% RSLogix 500 project TestPLC.RSS, saved by version 9.00.00.04 %
PROJECT "UNTITLED"    % processor: MicroLogix 1400 %

PROGRAM FILES
  LAD 2   17 rungs

DATA FILES
  O0 OUTPUT  6 elements
  I1 INPUT  8 elements
  S2 STATUS  66 elements
  B3 BINARY  3 elements
  T4 TIMER  3 elements
  C5 COUNTER  1 elements
  R6 CONTROL  1 elements
  N7 INTEGER  10 elements
  F8 FLOAT  3 elements
  N9 BATCH  11 elements  % store btch numbers %
  RI10   1 elements
  MG11 CREATESOCK  2 elements
  MG13   1 elements
  RI14   1 elements
  RI40   15 elements

LADDER 2
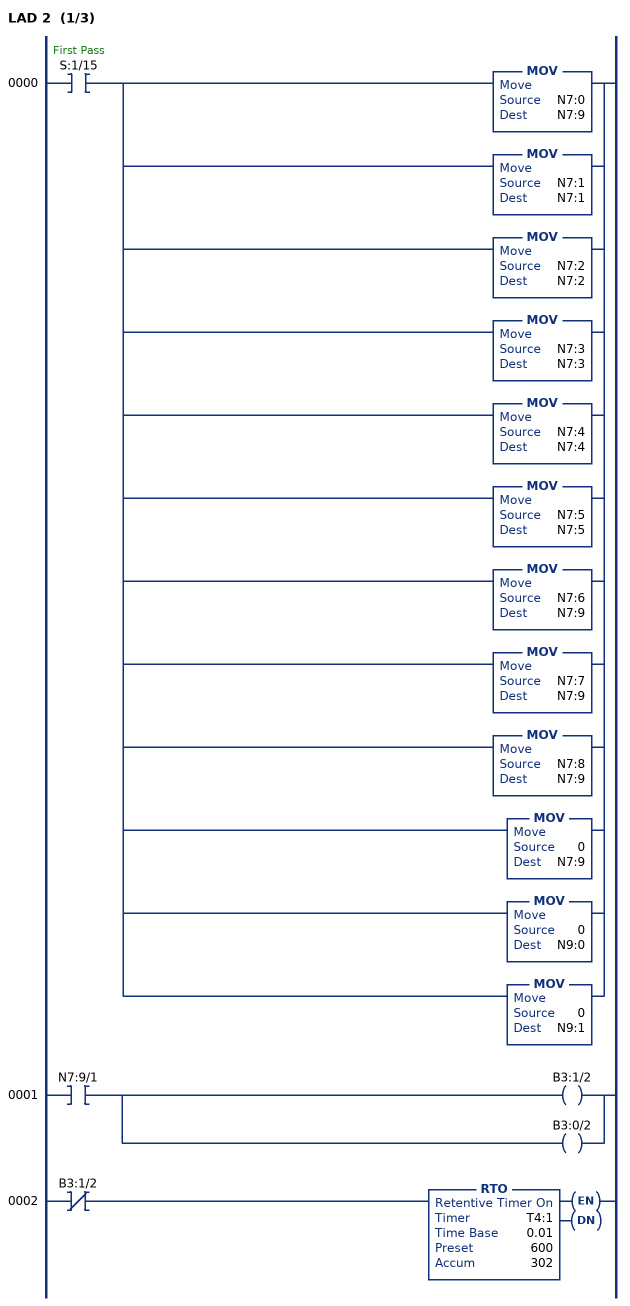
% Rung: 0 %
SOR XIC S:1/15 BST MOV N7:0 N7:9 NXB MOV N7:1 N7:1 NXB MOV N7:2 N7:2 NXB MOV N7:3 N7:3 NXB MOV N7:4 N7:4 NXB MOV N7:5 N7:5 NXB MOV N7:6 N7:9 NXB MOV N7:7 N7:9 NXB MOV N7:8 N7:9 NXB MOV 0 N7:9 NXB MOV 0 N9:0 NXB MOV 0 N9:1 BND EOR
%   S:1/15  "First Pass" %
%   N7:0  "Clr Control Block" %
% Rung: 1 %
SOR XIC N7:9/1 BST OTE B3:1/2 NXB OTE B3:0/2 BND EOR
% Rung: 2 %
SOR XIO B3:1/2 RTO T4:1 0.01 600 302 EOR

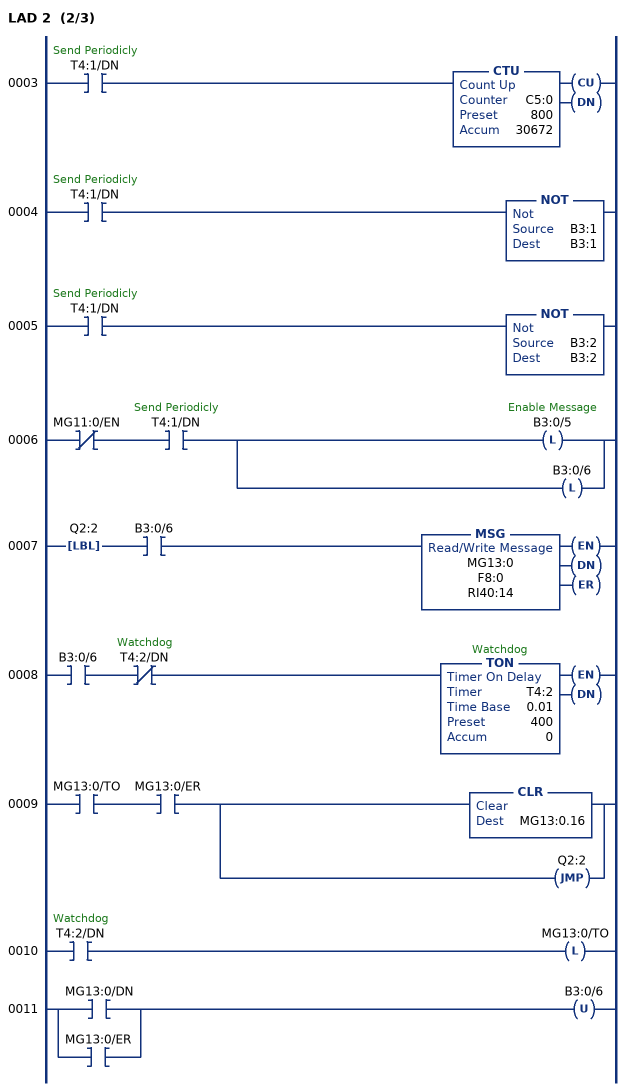
% Rung: 3 %
SOR XIC T4:1/DN CTU C5:0 800 30672 EOR
%   T4:1/DN  "Send Periodicly" %
% Rung: 4 %
SOR XIC T4:1/DN NOT B3:1 B3:1 EOR
%   T4:1/DN  "Send Periodicly" %
% Rung: 5 %
SOR XIC T4:1/DN NOT B3:2 B3:2 EOR
%   T4:1/DN  "Send Periodicly" %
% Rung: 6 %
SOR XIO MG11:0/EN XIC T4:1/DN BST OTL B3:0/5 NXB OTL B3:0/6 BND EOR
%   T4:1/DN  "Send Periodicly" %
%   B3:0/5  "Enable Message" %
% Rung: 7 %
SOR LBL Q2:2 XIC B3:0/6 MSG MG13:0 F8:0 RI40:14 EOR
%   MSG set-up: 500CPU Write | 33 | 2 | F8:7 | F8:0 | 0 | 0 | 0 | 192.168.1.10 | 0 | 0 | 192.168.1.10 | RI40:14 %
% Rung: 8 %
SOR XIC B3:0/6 XIO T4:2/DN TON T4:2 0.01 400 0 EOR
%   T4:2  "Watchdog" %
% Rung: 9 %
SOR XIC MG13:0/TO XIC MG13:0/ER BST CLR MG13:0.16 NXB JMP Q2:2 BND EOR
% Rung: 10 %
SOR XIC T4:2/DN OTL MG13:0/TO EOR
%   T4:2  "Watchdog" %
% Rung: 11 %
SOR BST XIC MG13:0/DN NXB XIC MG13:0/ER BND OTU B3:0/6 EOR

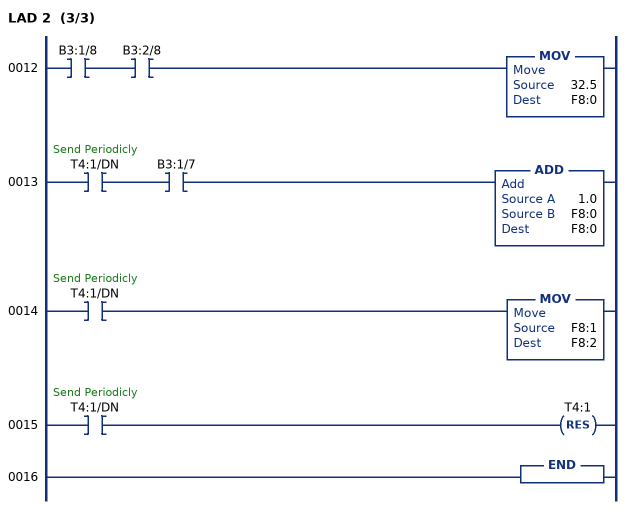
% Rung: 12 %
SOR XIC B3:1/8 XIC B3:2/8 MOV 32.5 F8:0 EOR
% Rung: 13 %
SOR XIC T4:1/DN XIC B3:1/7 ADD 1.0 F8:0 F8:0 EOR
%   T4:1/DN  "Send Periodicly" %
% Rung: 14 %
SOR XIC T4:1/DN MOV F8:1 F8:2 EOR
%   T4:1/DN  "Send Periodicly" %
% Rung: 15 %
SOR XIC T4:1/DN RES T4:1 EOR
%   T4:1/DN  "Send Periodicly" %
% Rung: 16 %
SOR END EOR

OTHER DOCUMENTED ADDRESSES
  B3:10  "Get Socket Instance"
  MG11:0.16  "Control"
  MG11:0.16/8  "TimeOut"
  MG11:0.17/12  "Error"
  MG11:0.17/13  "Msg Done"
  MG11:0/0  MG11
  N7:0/8  "TimeOut"
  N7:0/12  "Error"
  N7:10/0  "Instance number"
  Q2:1  "Try again"
  T4:0  "WatchDog"

COMMENTS NOT ATTACHED TO A CURRENT RUNG
  B3:10/0: Check periodically for socket instance number.

DATA TABLE (non-zero values as saved)
DATA B3
% B3:0 % 0XFFBB 0XFEEB 0XFFF9
DATA T4
% .PRE .ACC %
% T4:0 % 400 0
% T4:1 % 600 302
% T4:2 % 400 0
DATA C5
% .PRE .ACC %
% C5:0 % 800 30672
DATA N7
% N7:0 % 0 0 8888 9999 0 0 0 0 0 0
DATA F8
% F8:0 % 15706.5 65.5 65.5
DATA N9
% N9:0 % 0 0 3333 666 0 0 0 0 0 0
